(* IEC 61131-3 sources: verifaps-lib/geteta/examples/detwait, 3 files *)

(* ---- detwait.st ---- *)
PROGRAM dw
VAR_INPUT  i:INT; END_VAR
VAR_OUTPUT o:INT; END_VAR
VAR s : INT; END_VAR

s := s + 1;

IF i = 1 THEN
    o := 1;
ELSE
    o := s;
END_IF

END_PROGRAM

(* ---- detwait_long.st ---- *)
PROGRAM dw
VAR_INPUT  i:INT; END_VAR
VAR_OUTPUT o:INT; END_VAR
VAR s : INT; END_VAR

IF i = 0 THEN
    s := 0;
ELSEIF i > 0 THEN
    s := s + 1;
END_IF
o := s;
END_PROGRAM

(* ---- detwait_wrong.st ---- *)
PROGRAM dw
VAR_INPUT  i:INT; END_VAR
VAR_OUTPUT o:INT; END_VAR
VAR s : INT; END_VAR

s := s + 1;
o := s;

END_PROGRAM
